TYPE FireParameters :
STRUCT
	EN: BOOL := FALSE; // Run fan when FIRE
	Speed: LREAL := 0; // Speed when in FIRE (0-1)
END_STRUCT
END_TYPE

(* stored: Version 1.1.0.1, ProductVersion 3.1.4024.6
   DUT FireParameters: Id {6089c3e6-fe52-40a5-ac9e-036d207d68e3} *)
